{attribute 'qualified_only'}
VAR_GLOBAL
	STS : ARRAY [1..10] OF RTU_STS;
END_VAR

(* stored: Version 1.1.0.1, ProductVersion 3.1.4024.12
   GVL GVL_STS: Id {d83fe3ac-b354-4e29-8096-4b635bae75c0} *)
